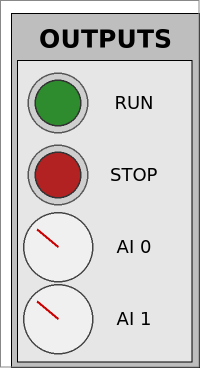
VISUALIZATION Dashboard  // 200x368
    RoundedRectangle (11,13 189x355)
    RoundedRectangle (17,60 175x302)
    Lamp1 (23,68 70x70), variable: GVL.DO0, style: Lamp-Lamp1-Green
    Lamp1 (23,140 70x70), variable: GVL.DO1, style: Lamp-Lamp1-Red
    Meter360 (23,284 70x70), value: GVL.AI1, style: Meter-Meter360-Gray, scale 0..20000
    Meter360 (23,212 70x70), value: GVL.AI1, style: Meter-Meter360-Gray, scale 0..20000
    Label (19,5 173x67), "OUTPUTS"
    Label (100,140 68x70), "STOP"
    Label (100,68 68x70), "RUN"
    Label (100,212 68x70), "AI 0"
    Label (100,284 68x70), "AI 1"
END_VISUALIZATION

(* stored: Version 1.1.0.1, ProductVersion 3.1.4024.12
   Visu Dashboard: Id {171ecf43-2f1b-4843-a75e-9636427ad08c} *)
